{attribute 'qualified_only'}
{attribute 'strict'}
TYPE E_ProcessCylinder_State :
(
		//GENERIC
	ABORTED				:=10,
	RESET_ERROR			:=20,
	HOMING				:=30,
	READY				:=40,
	//MANUAL_MODE			:=50, /manual mode not needed.
	ERROR				:=60,
	PERSISTENT_ERROR	:=70,
	STOPPING			:=80,
	//SPECIFIC FOR EVERY STATION
	Exntend				:=100,
	Retract				:=120,
	DONE				:=140,
	RESULTS				:=160,
	RESET				:=180
);
END_TYPE

(* stored: Version 1.1.0.1, ProductVersion 3.1.4024.13
   DUT E_ProcessCylinder_State: Id {39ea7c49-57ae-4672-9d34-1fe246bace50} *)
